// TIA Portal project "步进控制" (V20)

(* hardware
DEVICE "S7-1200 station_1"  S7-1200 Station
   slot 0: "Rack_0"  S7-1200 Rack  Rack  V1.0
   slot 1: "PLC_1"  CPU 1215C DC/DC/DC  6ES7 215-1AG40-0XB0  V4.6
   slot 3: "CB 1241 (RS485)"  CB 1241 (RS485)  6ES7 241-1CH30-1XB0  V1.0
*)

// ===== PLC "PLC_1"  CPU 1215C DC/DC/DC =====

VAR_GLOBAL   // PLC tag table "Default tag table"
   "桌面丝杆_Pulse" AT %Q0.0 : Bool;
   "桌面丝杆_Direction" AT %Q0.2 : Bool;
   "桌面丝杆_LowHwLimitSwitch" AT %I0.0 : Bool;
   "桌面丝杆_HighHwLimitSwitch" AT %I0.2 : Bool;
   "桌面丝杆_Homing switch" AT %I0.1 : Bool;
   "Tag_1" AT %I0.3 : Bool;
   "Tag_2" AT %Q0.1 : Bool;
   "Tag_3" AT %Q0.3 : Bool;
   "Tag_4" AT %Q0.4 : Bool;
   "Tag_5" AT %Q0.5 : Bool;
   "Tag_6" AT %Q0.6 : Bool;
   "Tag_7" AT %Q0.7 : Bool;
   "Tag_8" AT %Q1.0 : Bool;
   "Tag_9" AT %Q1.1 : Bool;
   "Tag_10" AT %Q1.2 : Bool;
   "Tag_11" AT %Q1.3 : Bool;
   "Tag_12" AT %Q1.4 : Bool;
   "Tag_13" AT %Q1.5 : Bool;
   "Tag_14" AT %Q1.6 : Bool;
   "Tag_15" AT %Q1.7 : Bool;
   "Tag_16" AT %Q2.0 : Bool;
   "Tag_17" AT %Q2.1 : Bool;
   "Tag_18" AT %Q2.2 : Bool;
   "Tag_19" AT %Q2.3 : Bool;
   "Tag_20" AT %Q2.4 : Bool;
   "Tag_21" AT %Q2.5 : Bool;
   "Tag_22" AT %Q2.6 : Bool;
   "Tag_23" AT %Q2.7 : Bool;
END_VAR

DATA_BLOCK "Block_1_DB"   // DB2
{ S7_Optimized_Access := 'FALSE' }
VERSION : 0.1
// stored: InstanceOfName Block_1
"Block_1"
BEGIN
END_DATA_BLOCK

DATA_BLOCK "Db Global"   // DB3
{ S7_Optimized_Access := 'TRUE' }
VERSION : 0.1
   VAR
      connection : TCON_IP_v4;
   END_VAR
BEGIN
   connection.InterfaceId := 64;
   connection.ID := 1;
   connection.LocalPort := 502;
END_DATA_BLOCK

DATA_BLOCK "ToDaxis_move_DB"   // DB5
{ S7_Optimized_Access := 'TRUE' }
VERSION : 0.1
// stored: InstanceOfName ToDaxis_move
"ToDaxis_move"
BEGIN
END_DATA_BLOCK

DATA_BLOCK "桌面丝杆"   // DB1, Motion_DB
{ S7_Optimized_Access := 'TRUE' }
AUTHOR : SIMATIC
FAMILY : BasicMC
NAME : TO_PosAx
VERSION : 8.0
// stored: InstanceOfName TO_PositioningAxis
"TO_PositioningAxis"
BEGIN
   // Axis.HomingReferencePointSwitch_AddressCU = %I0.1
   // Axis.LengthUnitNormalized.Distance = 1013
   // Axis.PositionLimitsMax_AddressCU = %I0.2
   // Axis.PositionLimitsMin_AddressCU = %I0.0
   // Axis.DirectionOutputEnabledCU = TRUE
   // Axis.OnlinePtoModeCU = 16#0000_0002
   // Axis.SelectedChannel2EnumCU = %Q0.2
   // Axis.SelectedChannel1EnumCU = %Q0.0
   // Pulse.MinDeltaDeltaFrequencyCU = 0.004
   // Pulse.MaxDeltaDeltaFrequencyCU = 1.0E+10
   // Pulse.MinDeltaFrequencyCU = 0.005
   // Pulse.MaxDeltaFrequencyCU = 9.5E+9
   // Pulse.MinFrequencyCU = 1.0
   // Pulse.MaxFrequencyCU = 100000.0
   // Pulse.OutputSourceCU = 16#0000_0000
   // Axis.SelectPTO = 0
END_DATA_BLOCK

FUNCTION_BLOCK "ToDaxis_move"   // FB1, LAD
{ S7_Optimized_Access := 'TRUE' }
VERSION : 0.1
   VAR
      regplace : DWord;
      connect_party : DWord;
      "step" : Int;
      start : Bool;
      confirmed : Bool;
      needconfirm : Bool;
      c_position : Real;
      return_position : Real;
      MC_Power_Instance : MC_Power;
      MC_Reset_Instance : MC_Reset;
      MC_Home_Instance : MC_Home;
      MC_Halt_Instance : MC_Halt;
      MC_MoveAbsolute_Instance : MC_MoveAbsolute;
      MC_MoveRelative_Instance : MC_MoveRelative;
      MC_MoveJog_Instance : MC_MoveJog;
      MC_MoveVelocity_Instance : MC_MoveVelocity;
      cache : Array[0..10] of Bool;
      cliping : Bool;
      t0 : TON_TIME;
      t1 : TON_TIME;
      t2 : TON_TIME;
   END_VAR
   VAR_TEMP   // added for the SCL form of the ladder/FBD networks
      _w1 : Bool;
      _w2 : Bool;
   END_VAR
BEGIN

REGION Network 1
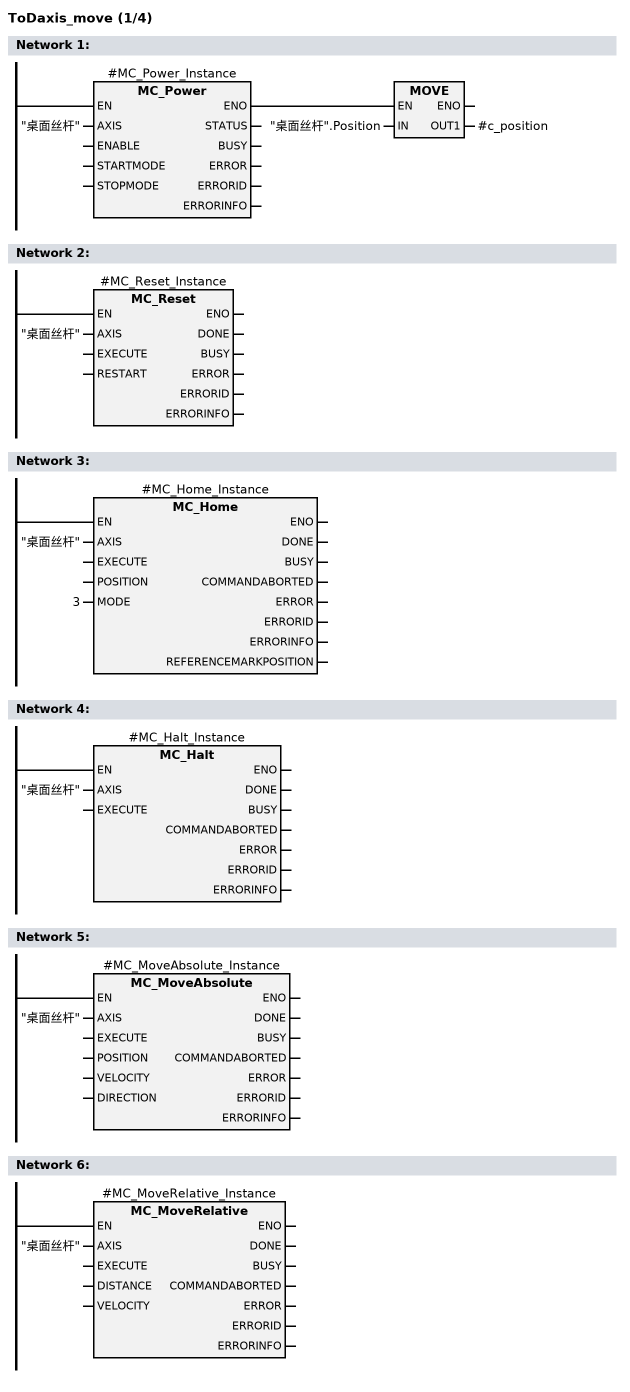
   // ENO of a box is taken as its EN; it also drops when the box reports an error
   #MC_Power_Instance(Axis := "桌面丝杆");   // MC_Power
   #c_position := "桌面丝杆".Position;
END_REGION

REGION Network 2
   #MC_Reset_Instance(Axis := "桌面丝杆");   // MC_Reset
END_REGION

REGION Network 3
   #MC_Home_Instance(Axis := "桌面丝杆", Mode := 3);   // MC_Home
END_REGION

REGION Network 4
   #MC_Halt_Instance(Axis := "桌面丝杆");   // MC_Halt
END_REGION

REGION Network 5
   #MC_MoveAbsolute_Instance(Axis := "桌面丝杆");   // MC_MoveAbsolute
END_REGION

REGION Network 6
   #MC_MoveRelative_Instance(Axis := "桌面丝杆");   // MC_MoveRelative
END_REGION

REGION Network 7
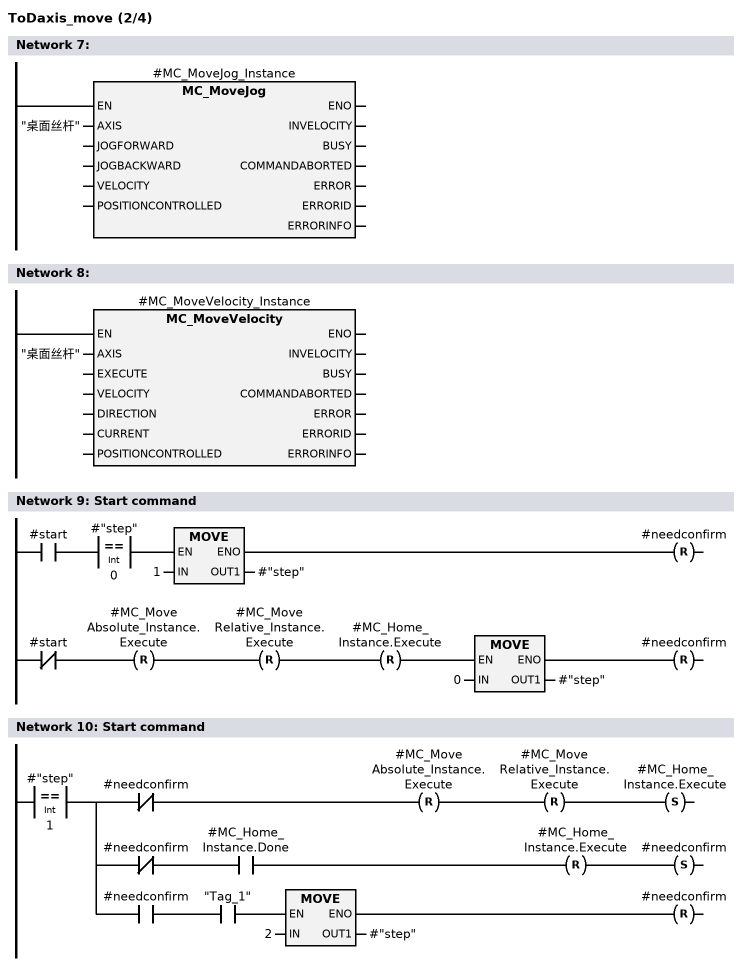
   #MC_MoveJog_Instance(Axis := "桌面丝杆");   // MC_MoveJog
END_REGION

REGION Network 8
   #MC_MoveVelocity_Instance(Axis := "桌面丝杆");   // MC_MoveVelocity
END_REGION

REGION Network 9: Start command
   RUNG wire#powerrail
      Contact( #start )
      { S7_Templates := "SrcType := Int" } EQ_Contact(in1 := #"step", in2 := 0)
      Move(in := 1, out1 => #"step")
      R_Coil( #needconfirm )
   END_RUNG
   RUNG wire#powerrail
      I_Contact( #start )
      R_Coil( #MC_MoveAbsolute_Instance.Execute )
      R_Coil( #MC_MoveRelative_Instance.Execute )
      R_Coil( #MC_Home_Instance.Execute )
      Move(in := 0, out1 => #"step")
      R_Coil( #needconfirm )
   END_RUNG
   // the same network as SCL:
   #_w1 := #start AND (#"step" = 0);
   IF #_w1 THEN
       #"step" := 1;
       #needconfirm := FALSE;
   END_IF;
   IF NOT #start THEN
       #MC_MoveAbsolute_Instance.Execute := FALSE;
       #MC_MoveRelative_Instance.Execute := FALSE;
       #MC_Home_Instance.Execute := FALSE;
       #"step" := 0;
       #needconfirm := FALSE;
   END_IF;
END_REGION

REGION Network 10: Start command
   RUNG wire#powerrail
      { S7_Templates := "SrcType := Int" } EQ_Contact(in1 := #"step", in2 := 1)
      wire#w1
      I_Contact( #needconfirm )
      R_Coil( #MC_MoveAbsolute_Instance.Execute )
      R_Coil( #MC_MoveRelative_Instance.Execute )
      S_Coil( #MC_Home_Instance.Execute )
   END_RUNG
   RUNG wire#w1
      I_Contact( #needconfirm )
      Contact( #MC_Home_Instance.Done )
      R_Coil( #MC_Home_Instance.Execute )
      S_Coil( #needconfirm )
   END_RUNG
   RUNG wire#w1
      Contact( #needconfirm )
      Contact( "Tag_1" )
      Move(in := 2, out1 => #"step")
      R_Coil( #needconfirm )
   END_RUNG
   // the same network as SCL:
   #_w1 := #"step" = 1;
   IF #_w1 AND NOT #needconfirm THEN
       #MC_MoveAbsolute_Instance.Execute := FALSE;
       #MC_MoveRelative_Instance.Execute := FALSE;
       #MC_Home_Instance.Execute := TRUE;
   END_IF;
   IF #_w1 AND NOT #needconfirm AND #MC_Home_Instance.Done THEN
       #MC_Home_Instance.Execute := FALSE;
       #needconfirm := TRUE;
   END_IF;
   IF #_w1 AND #needconfirm AND "Tag_1" THEN
       #"step" := 2;
       #needconfirm := FALSE;
   END_IF;
END_REGION

REGION Network 11: Start command
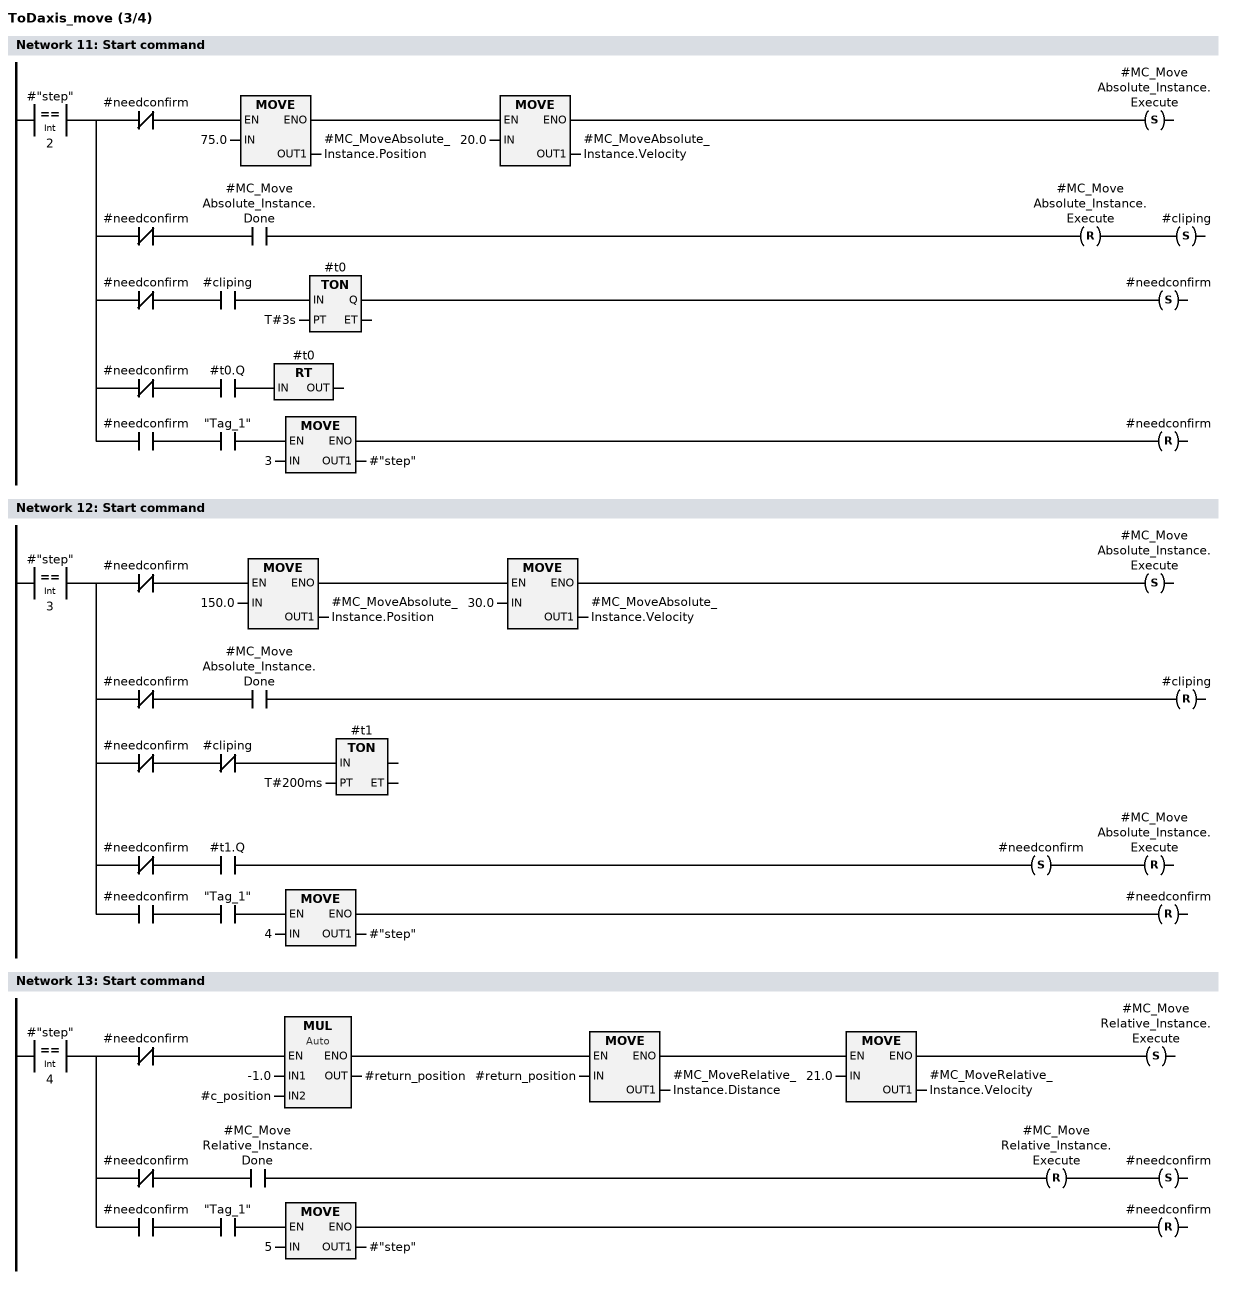
   #_w1 := #"step" = 2;
   IF #_w1 AND NOT #needconfirm THEN
       #MC_MoveAbsolute_Instance.Position := 75.0;
       #MC_MoveAbsolute_Instance.Velocity := 20.0;
       #MC_MoveAbsolute_Instance.Execute := TRUE;
   END_IF;
   IF #_w1 AND NOT #needconfirm AND #MC_MoveAbsolute_Instance.Done THEN
       #MC_MoveAbsolute_Instance.Execute := FALSE;
       #cliping := TRUE;
   END_IF;
   #t0(IN := #_w1 AND NOT #needconfirm AND #cliping, PT := T#3s);   // TON
   IF #t0.Q THEN #needconfirm := TRUE; END_IF;
   IF #_w1 AND NOT #needconfirm AND #t0.Q THEN RESET_TIMER(#t0); END_IF;
   IF #_w1 AND #needconfirm AND "Tag_1" THEN
       #"step" := 3;
       #needconfirm := FALSE;
   END_IF;
END_REGION

REGION Network 12: Start command
   #_w1 := #"step" = 3;
   IF #_w1 AND NOT #needconfirm THEN
       #MC_MoveAbsolute_Instance.Position := 150.0;
       #MC_MoveAbsolute_Instance.Velocity := 30.0;
       #MC_MoveAbsolute_Instance.Execute := TRUE;
   END_IF;
   IF #_w1 AND NOT #needconfirm AND #MC_MoveAbsolute_Instance.Done THEN #cliping := FALSE; END_IF;
   #t1(IN := #_w1 AND NOT #needconfirm AND NOT #cliping, PT := T#200ms);   // TON
   #_w2 := #_w1 AND NOT #needconfirm AND #t1.Q;
   IF #_w2 THEN
       #needconfirm := TRUE;
       #MC_MoveAbsolute_Instance.Execute := FALSE;
   END_IF;
   IF #_w1 AND #needconfirm AND "Tag_1" THEN
       #"step" := 4;
       #needconfirm := FALSE;
   END_IF;
END_REGION

REGION Network 13: Start command
   RUNG wire#powerrail
      { S7_Templates := "SrcType := Int" } EQ_Contact(in1 := #"step", in2 := 4)
      wire#w1
      I_Contact( #needconfirm )
      Mul(in1 := -1.0, in2 := #c_position, out => #return_position)
      Move(in := #return_position, out1 => #MC_MoveRelative_Instance.Distance)
      Move(in := 21.0, out1 => #MC_MoveRelative_Instance.Velocity)
      S_Coil( #MC_MoveRelative_Instance.Execute )
   END_RUNG
   RUNG wire#w1
      I_Contact( #needconfirm )
      Contact( #MC_MoveRelative_Instance.Done )
      R_Coil( #MC_MoveRelative_Instance.Execute )
      S_Coil( #needconfirm )
   END_RUNG
   RUNG wire#w1
      Contact( #needconfirm )
      Contact( "Tag_1" )
      Move(in := 5, out1 => #"step")
      R_Coil( #needconfirm )
   END_RUNG
   // the same network as SCL:
   #_w1 := #"step" = 4;
   IF #_w1 AND NOT #needconfirm THEN
       #return_position := (-1.0) * #c_position;
       #MC_MoveRelative_Instance.Distance := #return_position;
       #MC_MoveRelative_Instance.Velocity := 21.0;
       #MC_MoveRelative_Instance.Execute := TRUE;
   END_IF;
   IF #_w1 AND NOT #needconfirm AND #MC_MoveRelative_Instance.Done THEN
       #MC_MoveRelative_Instance.Execute := FALSE;
       #needconfirm := TRUE;
   END_IF;
   IF #_w1 AND #needconfirm AND "Tag_1" THEN
       #"step" := 5;
       #needconfirm := FALSE;
   END_IF;
END_REGION

REGION Network 14: Start command
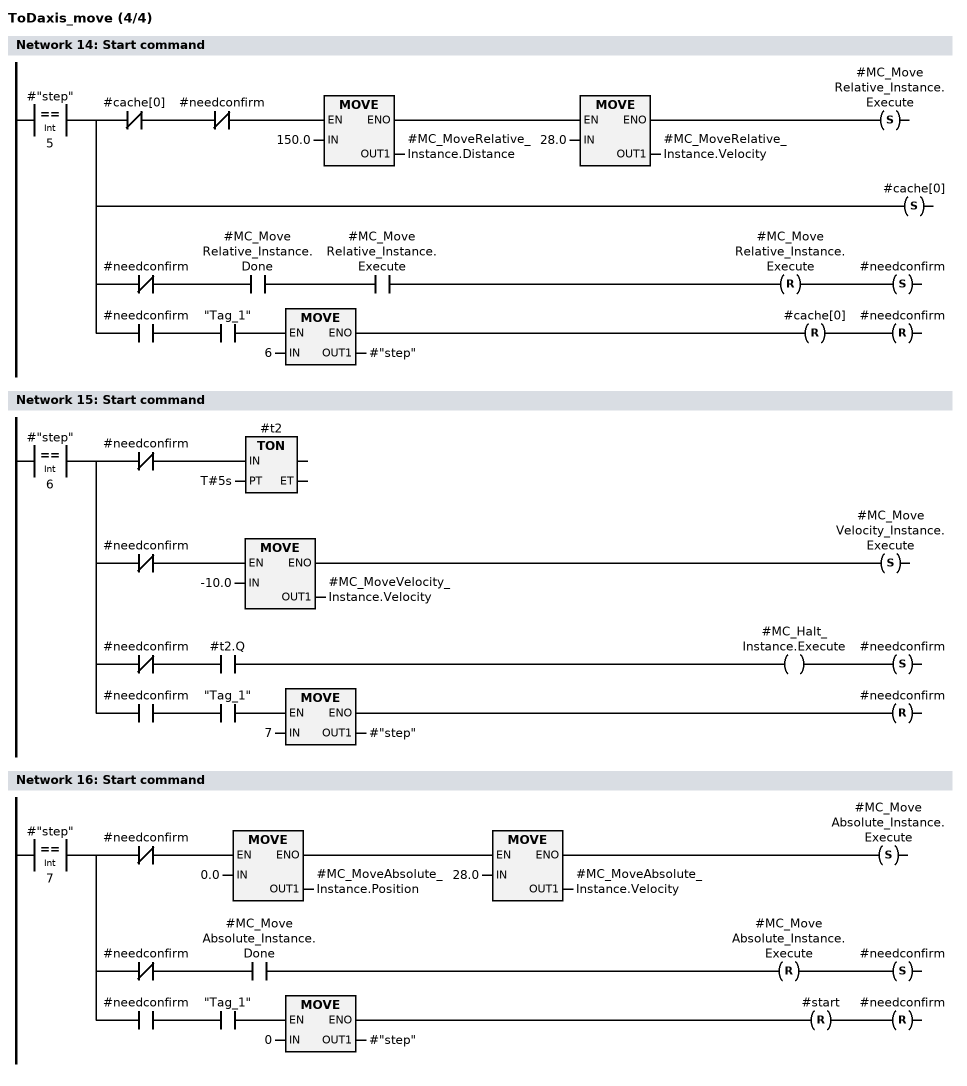
   RUNG wire#powerrail
      { S7_Templates := "SrcType := Int" } EQ_Contact(in1 := #"step", in2 := 5)
      wire#w1
      I_Contact( #cache[0] )
      I_Contact( #needconfirm )
      Move(in := 150.0, out1 => #MC_MoveRelative_Instance.Distance)
      Move(in := 28.0, out1 => #MC_MoveRelative_Instance.Velocity)
      S_Coil( #MC_MoveRelative_Instance.Execute )
   END_RUNG
   RUNG wire#w1
      S_Coil( #cache[0] )
   END_RUNG
   RUNG wire#w1
      I_Contact( #needconfirm )
      Contact( #MC_MoveRelative_Instance.Done )
      Contact( #MC_MoveRelative_Instance.Execute )
      R_Coil( #MC_MoveRelative_Instance.Execute )
      S_Coil( #needconfirm )
   END_RUNG
   RUNG wire#w1
      Contact( #needconfirm )
      Contact( "Tag_1" )
      Move(in := 6, out1 => #"step")
      R_Coil( #cache[0] )
      R_Coil( #needconfirm )
   END_RUNG
   // the same network as SCL:
   #_w1 := #"step" = 5;
   IF #_w1 AND NOT #cache[0] AND NOT #needconfirm THEN
       #MC_MoveRelative_Instance.Distance := 150.0;
       #MC_MoveRelative_Instance.Velocity := 28.0;
       #MC_MoveRelative_Instance.Execute := TRUE;
   END_IF;
   IF #_w1 THEN #cache[0] := TRUE; END_IF;
   #_w2 := #_w1 AND NOT #needconfirm AND #MC_MoveRelative_Instance.Done AND #MC_MoveRelative_Instance.Execute;
   IF #_w2 THEN
       #MC_MoveRelative_Instance.Execute := FALSE;
       #needconfirm := TRUE;
   END_IF;
   IF #_w1 AND #needconfirm AND "Tag_1" THEN
       #"step" := 6;
       #cache[0] := FALSE;
       #needconfirm := FALSE;
   END_IF;
END_REGION

REGION Network 15: Start command
   #_w1 := #"step" = 6;
   #t2(IN := #_w1 AND NOT #needconfirm, PT := T#5s);   // TON
   IF #_w1 AND NOT #needconfirm THEN
       #MC_MoveVelocity_Instance.Velocity := -10.0;
       #MC_MoveVelocity_Instance.Execute := TRUE;
   END_IF;
   #MC_Halt_Instance.Execute := #_w1 AND NOT #needconfirm AND #t2.Q;
   IF #MC_Halt_Instance.Execute THEN #needconfirm := TRUE; END_IF;
   IF #_w1 AND #needconfirm AND "Tag_1" THEN
       #"step" := 7;
       #needconfirm := FALSE;
   END_IF;
END_REGION

REGION Network 16: Start command
   RUNG wire#powerrail
      { S7_Templates := "SrcType := Int" } EQ_Contact(in1 := #"step", in2 := 7)
      wire#w1
      I_Contact( #needconfirm )
      Move(in := 0.0, out1 => #MC_MoveAbsolute_Instance.Position)
      Move(in := 28.0, out1 => #MC_MoveAbsolute_Instance.Velocity)
      S_Coil( #MC_MoveAbsolute_Instance.Execute )
   END_RUNG
   RUNG wire#w1
      I_Contact( #needconfirm )
      Contact( #MC_MoveAbsolute_Instance.Done )
      R_Coil( #MC_MoveAbsolute_Instance.Execute )
      S_Coil( #needconfirm )
   END_RUNG
   RUNG wire#w1
      Contact( #needconfirm )
      Contact( "Tag_1" )
      Move(in := 0, out1 => #"step")
      R_Coil( #start )
      R_Coil( #needconfirm )
   END_RUNG
   // the same network as SCL:
   #_w1 := #"step" = 7;
   IF #_w1 AND NOT #needconfirm THEN
       #MC_MoveAbsolute_Instance.Position := 0.0;
       #MC_MoveAbsolute_Instance.Velocity := 28.0;
       #MC_MoveAbsolute_Instance.Execute := TRUE;
   END_IF;
   IF #_w1 AND NOT #needconfirm AND #MC_MoveAbsolute_Instance.Done THEN
       #MC_MoveAbsolute_Instance.Execute := FALSE;
       #needconfirm := TRUE;
   END_IF;
   IF #_w1 AND #needconfirm AND "Tag_1" THEN
       #"step" := 0;
       #start := FALSE;
       #needconfirm := FALSE;
   END_IF;
END_REGION
END_FUNCTION_BLOCK

FUNCTION_BLOCK "Block_1"   // FB2, SCL
{ S7_Optimized_Access := 'FALSE' }
VERSION : 0.1
   VAR
      value1 : Word;
      value2 : Word;
      value3 : Word;
      value4 : Word;
      value5 : Word;
      value6 : Word;
      value7 : Word;
      value8 : Word;
      value9 : Word;
      value10 : Word;
      value11 : Word;
      value12 : Word;
      value13 : Word;
      value14 : Word;
      value15 : Word;
      value16 : Word;
      value17 : Word;
      value18 : Word;
      value19 : Word;
      value20 : Word;
      value21 : Word;
      value22 : Word;
      value23 : Word;
      value24 : Word;
      value25 : Word;
      value26 : Word;
      value27 : Word;
      value28 : Word;
      value29 : Word;
      value30 : Word;
   END_VAR
BEGIN
END_FUNCTION_BLOCK

ORGANIZATION_BLOCK "Main"   // OB1, LAD, ProgramCycle
TITLE = "Main Program Sweep (Cycle)"
{ S7_Optimized_Access := 'TRUE' }
VERSION : 0.1
   VAR_INPUT
      Initial_Call : Bool;   // Initial call of this OB
      Remanence : Bool;   // =True, if remanent data are available
   END_VAR
BEGIN

REGION Network 1
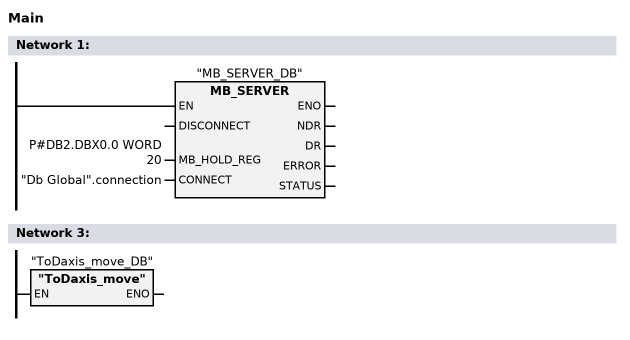
   "MB_SERVER_DB"(MB_HOLD_REG := P#DB2.DBX0.0 WORD 20, CONNECT := "Db Global".connection);   // MB_SERVER
END_REGION

REGION Network 3
   RUNG wire#powerrail
      "ToDaxis_move_DB"()
   END_RUNG
   // the same network as SCL:
   "ToDaxis_move_DB"();   // "ToDaxis_move"
END_REGION
END_ORGANIZATION_BLOCK